// TIA Portal V20 export
FUNCTION_BLOCK "FB_Digital_Inputs"   // FB1, LAD
{ S7_Optimized_Access := 'TRUE' }
// stored: MemoryReserve 100, SetENOAutomatically false
   VAR_INPUT
      I_Button_Start_Approve : Bool;
      I_Digital_Input_1 : Bool;
      I_Digital_Input_2 : Bool;
      I_Digital_Input_3 : Bool;
      I_Digital_Input_4 : Bool;
      I_Digital_Input_5 : Bool;
   END_VAR
   VAR_OUTPUT
      DB_Button_Start_Approve : Bool;
      DB_Digital_Input_1 : Bool;
      DB_Digital_Input_2 : Bool;
      DB_Digital_Input_3 : Bool;
      DB_Digital_Input_4 : Bool;
      DB_Digital_Input_5 : Bool;
   END_VAR
BEGIN

REGION Network 1
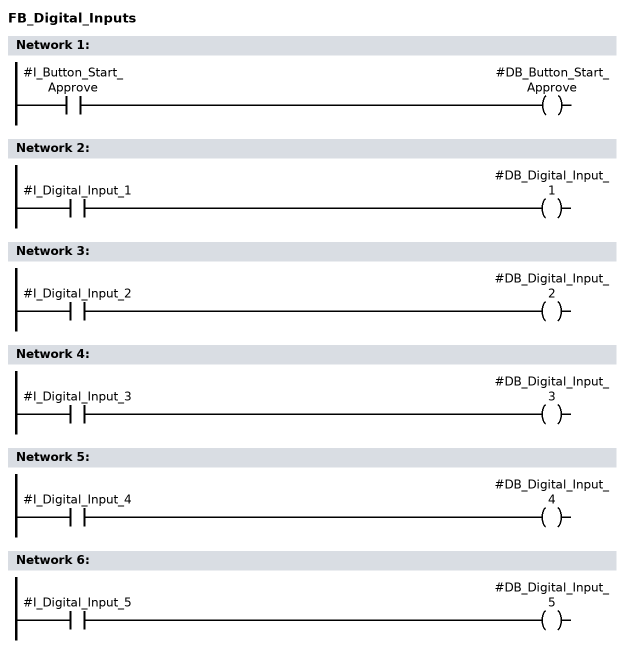
   RUNG wire#powerrail
      Contact( #I_Button_Start_Approve )
      Coil( #DB_Button_Start_Approve )
   END_RUNG
   // the same network as SCL:
   #DB_Button_Start_Approve := #I_Button_Start_Approve;
END_REGION

REGION Network 2
   RUNG wire#powerrail
      Contact( #I_Digital_Input_1 )
      Coil( #DB_Digital_Input_1 )
   END_RUNG
   // the same network as SCL:
   #DB_Digital_Input_1 := #I_Digital_Input_1;
END_REGION

REGION Network 3
   RUNG wire#powerrail
      Contact( #I_Digital_Input_2 )
      Coil( #DB_Digital_Input_2 )
   END_RUNG
   // the same network as SCL:
   #DB_Digital_Input_2 := #I_Digital_Input_2;
END_REGION

REGION Network 4
   RUNG wire#powerrail
      Contact( #I_Digital_Input_3 )
      Coil( #DB_Digital_Input_3 )
   END_RUNG
   // the same network as SCL:
   #DB_Digital_Input_3 := #I_Digital_Input_3;
END_REGION

REGION Network 5
   RUNG wire#powerrail
      Contact( #I_Digital_Input_4 )
      Coil( #DB_Digital_Input_4 )
   END_RUNG
   // the same network as SCL:
   #DB_Digital_Input_4 := #I_Digital_Input_4;
END_REGION

REGION Network 6
   RUNG wire#powerrail
      Contact( #I_Digital_Input_5 )
      Coil( #DB_Digital_Input_5 )
   END_RUNG
   // the same network as SCL:
   #DB_Digital_Input_5 := #I_Digital_Input_5;
END_REGION
END_FUNCTION_BLOCK
